% RSLogix 500 project Sensor-Calibration.RSS, saved by version 8.30.00.16 %
PROJECT "UNTITLED"    % processor: Bul.1763 MicroLogix 1100 Series B %

PROGRAM FILES
  LAD 2 "MAIN"  3 rungs
  LAD 3 "OUTPUT"  3 rungs
  LAD 4 "CTRL"  10 rungs

DATA FILES
  O0 OUTPUT  4 elements
  I1 INPUT  6 elements
  S2 STATUS  66 elements
  B3 BINARY  2 elements
  T4 TIMER  1 elements
  C5 COUNTER  1 elements
  R6 CONTROL  1 elements
  N7 INTEGER  7 elements
  F8 FLOAT  2 elements

LADDER 2 "MAIN"
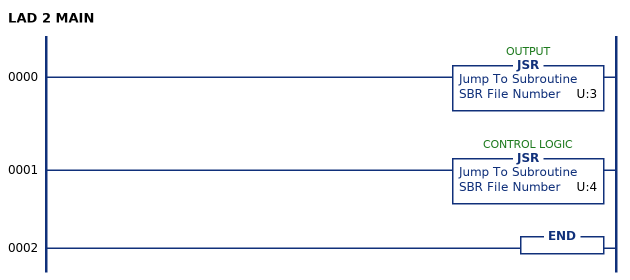
% Rung: 0 %
SOR JSR U:3 EOR
%   U:3  "OUTPUT" %
% Rung: 1 %
SOR JSR U:4 EOR
%   U:4  "CONTROL LOGIC" %
% Rung: 2 %
SOR END EOR

LADDER 3 "OUTPUT"
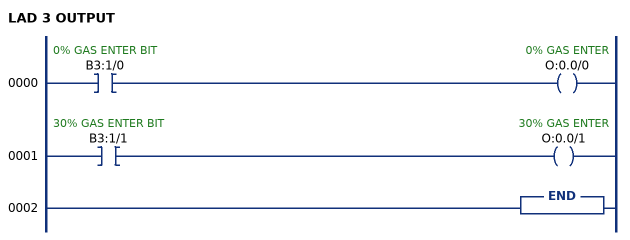
% Rung: 0 %
SOR XIC B3:1/0 OTE O:0.0/0 EOR
%   B3:1/0  "0% GAS ENTER BIT" %
%   O:0.0/0  "0% GAS ENTER" %
% Rung: 1 %
SOR XIC B3:1/1 OTE O:0.0/1 EOR
%   B3:1/1  "30% GAS ENTER BIT" %
%   O:0.0/1  "30% GAS ENTER" %
% Rung: 2 %
SOR END EOR

LADDER 4 "CTRL"
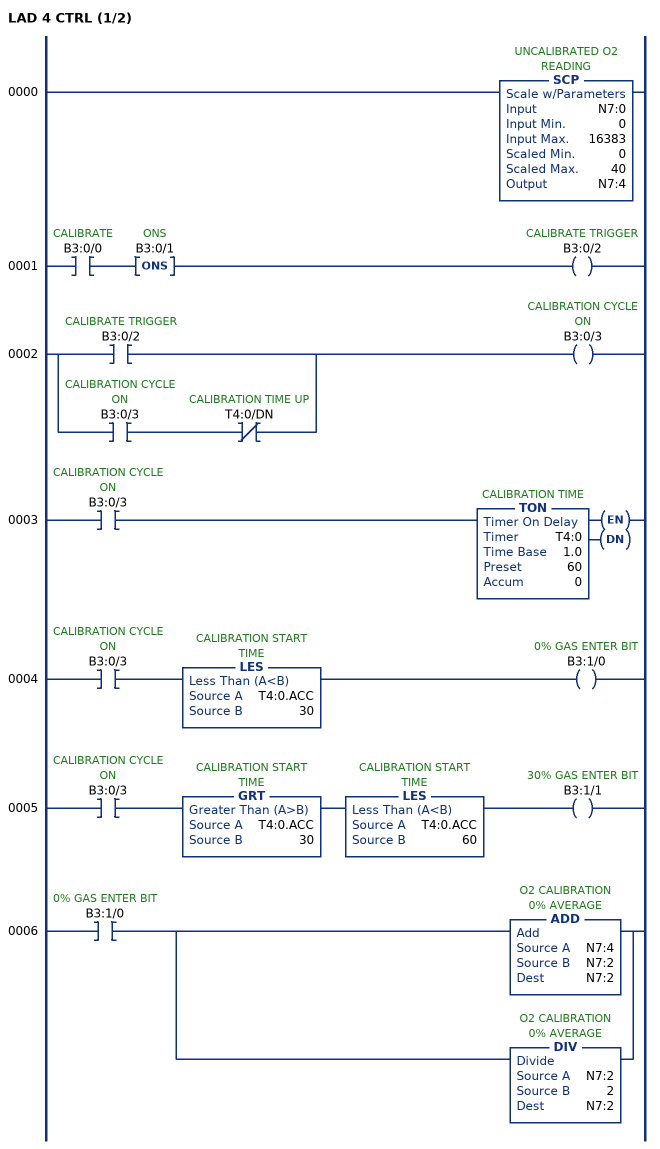
% Rung: 0 %
SOR SCP N7:0 0 16383 0 40 N7:4 EOR
%   N7:0  "O2 SENSOR INPUT" %
%   N7:4  "UNCALIBRATED O2 READING" %
% Rung: 1 %
SOR XIC B3:0/0 ONS B3:0/1 OTE B3:0/2 EOR
%   B3:0/0  "CALIBRATE" %
%   B3:0/1  "ONS" %
%   B3:0/2  "CALIBRATE TRIGGER" %
% Rung: 2 %
SOR BST XIC B3:0/2 NXB XIC B3:0/3 XIO T4:0/DN BND OTE B3:0/3 EOR
%   B3:0/2  "CALIBRATE TRIGGER" %
%   B3:0/3  "CALIBRATION CYCLE ON" %
%   T4:0/DN  "CALIBRATION TIME UP" %
% Rung: 3 %
SOR XIC B3:0/3 TON T4:0 1.0 60 0 EOR
%   B3:0/3  "CALIBRATION CYCLE ON" %
%   T4:0  "CALIBRATION TIME" %
% Rung: 4 %
SOR XIC B3:0/3 LES T4:0.ACC 30 OTE B3:1/0 EOR
%   B3:0/3  "CALIBRATION CYCLE ON" %
%   T4:0.ACC  "CALIBRATION START TIME" %
%   B3:1/0  "0% GAS ENTER BIT" %
% Rung: 5 %
SOR XIC B3:0/3 GRT T4:0.ACC 30 LES T4:0.ACC 60 OTE B3:1/1 EOR
%   B3:0/3  "CALIBRATION CYCLE ON" %
%   T4:0.ACC  "CALIBRATION START TIME" %
%   B3:1/1  "30% GAS ENTER BIT" %
% Rung: 6 %
SOR XIC B3:1/0 BST ADD N7:4 N7:2 N7:2 NXB DIV N7:2 2 N7:2 BND EOR
%   B3:1/0  "0% GAS ENTER BIT" %
%   N7:4  "UNCALIBRATED O2 READING" %
%   N7:2  "O2 CALIBRATION 0% AVERAGE" %

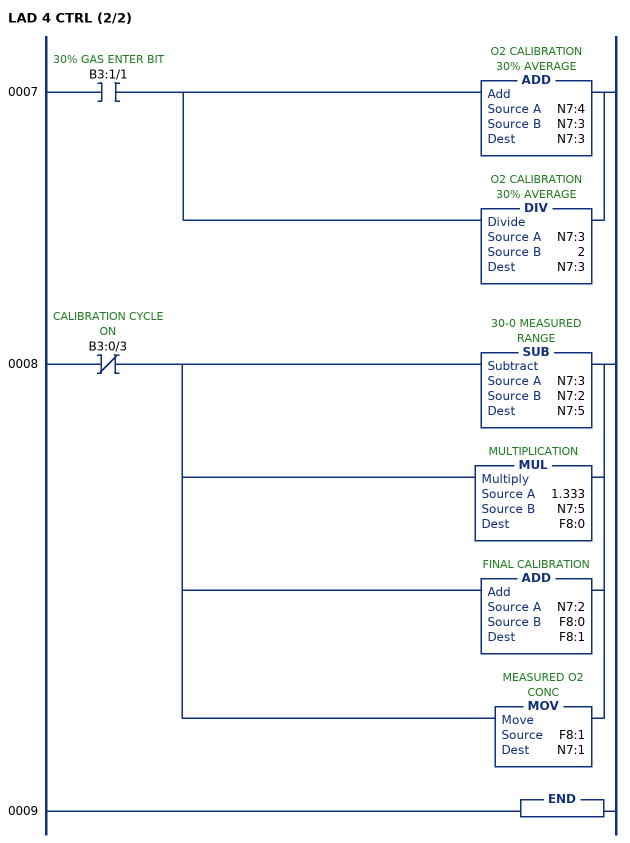
% Rung: 7 %
SOR XIC B3:1/1 BST ADD N7:4 N7:3 N7:3 NXB DIV N7:3 2 N7:3 BND EOR
%   B3:1/1  "30% GAS ENTER BIT" %
%   N7:4  "UNCALIBRATED O2 READING" %
%   N7:3  "O2 CALIBRATION 30% AVERAGE" %
% Rung: 8 %
SOR XIO B3:0/3 BST SUB N7:3 N7:2 N7:5 NXB BST MUL 1.333 N7:5 F8:0 NXB BST ADD N7:2 F8:0 F8:1 NXB MOV F8:1 N7:1 BND BND BND EOR
%   B3:0/3  "CALIBRATION CYCLE ON" %
%   N7:3  "O2 CALIBRATION 30% AVERAGE" %
%   N7:2  "O2 CALIBRATION 0% AVERAGE" %
%   N7:5  "30-0 MEASURED RANGE" %
%   F8:0  "MULTIPLICATION" %
%   F8:1  "FINAL CALIBRATION" %
%   N7:1  "MEASURED O2 CONC" %
% Rung: 9 %
SOR END EOR

OTHER DOCUMENTED ADDRESSES
  B3:0/4  "CALIBRATION TIMEUP"
  C5:0  "COUNT FOR 0% AVERAGE"
  N7:6  "CALIB STEP"

DATA TABLE (non-zero values as saved)
DATA T4
% .PRE .ACC %
% T4:0 % 60 0
DATA N7
% N7:0 % 0 0 0 30 0 0 0
